{region '#Template'}
	{attribute 'Version' := '5.0.0.0'}
	{attribute 'Tags' := '"LCID": "1031", "Text": "Universal, Object, AV"'}
	{attribute 'Tags' := '"LCID": "1033", "Text": "Universal, Sensor, AV"'}
	{attribute 'Using' := '"Type": "Template", "URI": "EC_ID"'}
	{attribute 'Using' := '"Type": "Template", "URI": "BA2_Param"'}
	{attribute 'Description' := '"LCID": "1031", "Text": "AV"'}
	{attribute 'Description' := '"LCID": "1033", "Text": "AV"'}
{endregion}
FUNCTION_BLOCK FB_BA_AV_Op_Val EXTENDS FB_BA_View
VAR_INPUT
	fIn					: REAL;
END_VAR
VAR_OUTPUT
	fPresentValue				: REAL;
END_VAR
VAR_INPUT CONSTANT
	Val					: FB_BA_AV_Op;		
END_VAR
VAR
END_VAR

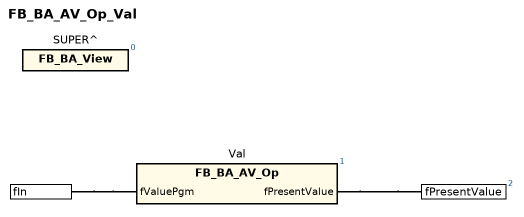
SUPER^(); // FB_BA_View
Val(fValuePgm := fIn); // FB_BA_AV_Op
fPresentValue := Val.fPresentValue;

METHOD FB_init : BOOL
VAR_INPUT
	bInitRetains : BOOL; // if TRUE, the retain variables are initialized (warm start / cold start)
	bInCopyCode : BOOL;  // if TRUE, the instance afterwards gets moved into the copy code (online change)
END_VAR
Val.iParent					:= THIS^;
Val.iLabel					:= LblFun_MeasuredValue;
Val.eUnit					:= E_BA_Unit.eTemperature_DegreesCelsius;  
Val.fCOVIncrement			:= BA2_Param.fDefCOVIncrement;
END_METHOD

END_FUNCTION_BLOCK

(* stored: Version 1.1.0.1, ProductVersion 3.1.4024.12
   POU FB_BA_AV_Op_Val: Id {acdf901d-16b4-4109-a63b-242b1b6b730e}, SpecialFunc None
   Method FB_init: Id {8deb770d-9ce3-4383-ac12-e565b73088ff} *)
